// TIA Portal V19 export
VAR_GLOBAL   // PLC tag table "Unit"
END_VAR
VAR_GLOBAL CONSTANT   // user constants
   NO_OF_EMs : Int := 2;   // Highest Value of equipment modules in the unit (Counting starts from 0)
   EM0 : Int := 0;   // Equipment Module 0
   EM1 : Int := 1;   // Equipment Module 1
   EM2 : Int := 2;   // Equipment Module 2
END_VAR
